(* IEC 61131-3 sources: AXOpen/src/io/app/SystemConstants, 2 files *)

(* ---- plc_line_IoAddresses.st ---- *)
CONFIGURATION IoAddresses
    VAR_GLOBAL

        // Module bnixg35080b5r067/IDM_LinkModule
        bnixg35080b5r067_IDM_LinkModule_BALLUFF_8_Port_IO_Link_Master_Input AT %IB0 : bnixg35080b5r067_IDM_LinkModule_BALLUFF_8_Port_IO_Link_Master_Input_Layout;
        bnixg35080b5r067_IDM_LinkModule_BALLUFF_8_Port_IO_Link_Master_Output AT %QB0 : bnixg35080b5r067_IDM_LinkModule_BALLUFF_8_Port_IO_Link_Master_Output_Layout;
        bnixg35080b5r067_IDM_LinkModule_X01_Input AT %IB1 : bnixg35080b5r067_IDM_LinkModule_X01_Input_Layout;

        // Module et200sp_1/A10
        et200sp_1_A10_Input AT %IB28 : et200sp_1_A10_Input_Layout;

        // Module et200sp_1/A11
        et200sp_1_A11_Input AT %IB26 : et200sp_1_A11_Input_Layout;

        // Module et200sp_1/A12
        et200sp_1_A12_Input AT %IB24 : et200sp_1_A12_Input_Layout;

        // Module et200sp_1/A13
        et200sp_1_A13_Input AT %IB22 : et200sp_1_A13_Input_Layout;

        // Module et200sp_1/A14
        et200sp_1_A14_Input AT %IB20 : et200sp_1_A14_Input_Layout;

        // Module et200sp_1/A15
        et200sp_1_A15_Input AT %IB18 : et200sp_1_A15_Input_Layout;

        // Module et200sp_1/A16
        et200sp_1_A16_Input AT %IB16 : et200sp_1_A16_Input_Layout;

        // Module et200sp_1/A17
        et200sp_1_A17_Input AT %IB14 : et200sp_1_A17_Input_Layout;

        // Module et200sp_1/A20
        et200sp_1_A20_Output AT %QB15 : et200sp_1_A20_Output_Layout;

        // Module et200sp_1/A21
        et200sp_1_A21_Output AT %QB13 : et200sp_1_A21_Output_Layout;

        // Module et200sp_1/A22
        et200sp_1_A22_Output AT %QB11 : et200sp_1_A22_Output_Layout;

        // Module et200sp_1/A23
        et200sp_1_A23_Output AT %QB9 : et200sp_1_A23_Output_Layout;

        // Module et200sp_1/A30
        et200sp_1_A30_Input AT %IB6 : et200sp_1_A30_Input_Layout;

        // Module et200sp_1/A40
        et200sp_1_A40_Output AT %QB1 : et200sp_1_A40_Output_Layout;

        // Module et200sp/A10
        et200sp_A10_Input AT %IB62 : et200sp_A10_Input_Layout;

        // Module et200sp/A20
        et200sp_A20_Output AT %QB49 : et200sp_A20_Output_Layout;

        // Module et200sp/A30
        et200sp_A30_Input AT %IB30 : et200sp_A30_Input_Layout;
        et200sp_A30_Output AT %QB17 : et200sp_A30_Output_Layout;
    END_VAR
END_CONFIGURATION

TYPE
    bnixg35080b5r067_IDM_LinkModule_BALLUFF_8_Port_IO_Link_Master_Input_Layout : STRUCT
        Signals_0 AT %X0.0 : BOOL;
        Signals_1 AT %X0.1 : BOOL;
        Signals_2 AT %X0.2 : BOOL;
        Signals_3 AT %X0.3 : BOOL;
        Signals_4 AT %X0.4 : BOOL;
        Signals_5 AT %X0.5 : BOOL;
        Signals_6 AT %X0.6 : BOOL;
        Signals_7 AT %X0.7 : BOOL;
    END_STRUCT;
END_TYPE

TYPE
    bnixg35080b5r067_IDM_LinkModule_BALLUFF_8_Port_IO_Link_Master_Output_Layout : STRUCT
        Signals_8 AT %X0.0 : BOOL;
        Signals_9 AT %X0.1 : BOOL;
        Signals_10 AT %X0.2 : BOOL;
        Signals_11 AT %X0.3 : BOOL;
        Signals_12 AT %X0.4 : BOOL;
        Signals_13 AT %X0.5 : BOOL;
        Signals_14 AT %X0.6 : BOOL;
        Signals_15 AT %X0.7 : BOOL;
    END_STRUCT;
END_TYPE

TYPE
    bnixg35080b5r067_IDM_LinkModule_X01_Input_Layout : STRUCT
        Signals_0 AT %B0 : ARRAY[0..3] OF BYTE;
        Signals_1 AT %X4.2 : BOOL;
        Signals_2 AT %X4.3 : BOOL;
        Signals_3 AT %X4.4 : BOOL;
        Signals_4 AT %X4.5 : BOOL;
        Signals_5 AT %X4.6 : BOOL;
        Signals_6 AT %X4.7 : BOOL;
    END_STRUCT;
END_TYPE

TYPE
    et200sp_1_A10_Input_Layout : STRUCT
        Signals_0 AT %X0.0 : BOOL;
        Signals_1 AT %X0.1 : BOOL;
        Signals_2 AT %X0.2 : BOOL;
        Signals_3 AT %X0.3 : BOOL;
        Signals_4 AT %X0.4 : BOOL;
        Signals_5 AT %X0.5 : BOOL;
        Signals_6 AT %X0.6 : BOOL;
        Signals_7 AT %X0.7 : BOOL;
        Signals_8 AT %X1.0 : BOOL;
        Signals_9 AT %X1.1 : BOOL;
        Signals_10 AT %X1.2 : BOOL;
        Signals_11 AT %X1.3 : BOOL;
        Signals_12 AT %X1.4 : BOOL;
        Signals_13 AT %X1.5 : BOOL;
        Signals_14 AT %X1.6 : BOOL;
        Signals_15 AT %X1.7 : BOOL;
    END_STRUCT;
END_TYPE

TYPE
    et200sp_1_A11_Input_Layout : STRUCT
        Signals_0 AT %X0.0 : BOOL;
        Signals_1 AT %X0.1 : BOOL;
        Signals_2 AT %X0.2 : BOOL;
        Signals_3 AT %X0.3 : BOOL;
        Signals_4 AT %X0.4 : BOOL;
        Signals_5 AT %X0.5 : BOOL;
        Signals_6 AT %X0.6 : BOOL;
        Signals_7 AT %X0.7 : BOOL;
        Signals_8 AT %X1.0 : BOOL;
        Signals_9 AT %X1.1 : BOOL;
        Signals_10 AT %X1.2 : BOOL;
        Signals_11 AT %X1.3 : BOOL;
        Signals_12 AT %X1.4 : BOOL;
        Signals_13 AT %X1.5 : BOOL;
        Signals_14 AT %X1.6 : BOOL;
        Signals_15 AT %X1.7 : BOOL;
    END_STRUCT;
END_TYPE

TYPE
    et200sp_1_A12_Input_Layout : STRUCT
        Signals_0 AT %X0.0 : BOOL;
        Signals_1 AT %X0.1 : BOOL;
        Signals_2 AT %X0.2 : BOOL;
        Signals_3 AT %X0.3 : BOOL;
        Signals_4 AT %X0.4 : BOOL;
        Signals_5 AT %X0.5 : BOOL;
        Signals_6 AT %X0.6 : BOOL;
        Signals_7 AT %X0.7 : BOOL;
        Signals_8 AT %X1.0 : BOOL;
        Signals_9 AT %X1.1 : BOOL;
        Signals_10 AT %X1.2 : BOOL;
        Signals_11 AT %X1.3 : BOOL;
        Signals_12 AT %X1.4 : BOOL;
        Signals_13 AT %X1.5 : BOOL;
        Signals_14 AT %X1.6 : BOOL;
        Signals_15 AT %X1.7 : BOOL;
    END_STRUCT;
END_TYPE

TYPE
    et200sp_1_A13_Input_Layout : STRUCT
        Signals_0 AT %X0.0 : BOOL;
        Signals_1 AT %X0.1 : BOOL;
        Signals_2 AT %X0.2 : BOOL;
        Signals_3 AT %X0.3 : BOOL;
        Signals_4 AT %X0.4 : BOOL;
        Signals_5 AT %X0.5 : BOOL;
        Signals_6 AT %X0.6 : BOOL;
        Signals_7 AT %X0.7 : BOOL;
        Signals_8 AT %X1.0 : BOOL;
        Signals_9 AT %X1.1 : BOOL;
        Signals_10 AT %X1.2 : BOOL;
        Signals_11 AT %X1.3 : BOOL;
        Signals_12 AT %X1.4 : BOOL;
        Signals_13 AT %X1.5 : BOOL;
        Signals_14 AT %X1.6 : BOOL;
        Signals_15 AT %X1.7 : BOOL;
    END_STRUCT;
END_TYPE

TYPE
    et200sp_1_A14_Input_Layout : STRUCT
        Signals_0 AT %X0.0 : BOOL;
        Signals_1 AT %X0.1 : BOOL;
        Signals_2 AT %X0.2 : BOOL;
        Signals_3 AT %X0.3 : BOOL;
        Signals_4 AT %X0.4 : BOOL;
        Signals_5 AT %X0.5 : BOOL;
        Signals_6 AT %X0.6 : BOOL;
        Signals_7 AT %X0.7 : BOOL;
        Signals_8 AT %X1.0 : BOOL;
        Signals_9 AT %X1.1 : BOOL;
        Signals_10 AT %X1.2 : BOOL;
        Signals_11 AT %X1.3 : BOOL;
        Signals_12 AT %X1.4 : BOOL;
        Signals_13 AT %X1.5 : BOOL;
        Signals_14 AT %X1.6 : BOOL;
        Signals_15 AT %X1.7 : BOOL;
    END_STRUCT;
END_TYPE

TYPE
    et200sp_1_A15_Input_Layout : STRUCT
        Signals_0 AT %X0.0 : BOOL;
        Signals_1 AT %X0.1 : BOOL;
        Signals_2 AT %X0.2 : BOOL;
        Signals_3 AT %X0.3 : BOOL;
        Signals_4 AT %X0.4 : BOOL;
        Signals_5 AT %X0.5 : BOOL;
        Signals_6 AT %X0.6 : BOOL;
        Signals_7 AT %X0.7 : BOOL;
        Signals_8 AT %X1.0 : BOOL;
        Signals_9 AT %X1.1 : BOOL;
        Signals_10 AT %X1.2 : BOOL;
        Signals_11 AT %X1.3 : BOOL;
        Signals_12 AT %X1.4 : BOOL;
        Signals_13 AT %X1.5 : BOOL;
        Signals_14 AT %X1.6 : BOOL;
        Signals_15 AT %X1.7 : BOOL;
    END_STRUCT;
END_TYPE

TYPE
    et200sp_1_A16_Input_Layout : STRUCT
        Signals_0 AT %X0.0 : BOOL;
        Signals_1 AT %X0.1 : BOOL;
        Signals_2 AT %X0.2 : BOOL;
        Signals_3 AT %X0.3 : BOOL;
        Signals_4 AT %X0.4 : BOOL;
        Signals_5 AT %X0.5 : BOOL;
        Signals_6 AT %X0.6 : BOOL;
        Signals_7 AT %X0.7 : BOOL;
        Signals_8 AT %X1.0 : BOOL;
        Signals_9 AT %X1.1 : BOOL;
        Signals_10 AT %X1.2 : BOOL;
        Signals_11 AT %X1.3 : BOOL;
        Signals_12 AT %X1.4 : BOOL;
        Signals_13 AT %X1.5 : BOOL;
        Signals_14 AT %X1.6 : BOOL;
        Signals_15 AT %X1.7 : BOOL;
    END_STRUCT;
END_TYPE

TYPE
    et200sp_1_A17_Input_Layout : STRUCT
        Signals_0 AT %X0.0 : BOOL;
        Signals_1 AT %X0.1 : BOOL;
        Signals_2 AT %X0.2 : BOOL;
        Signals_3 AT %X0.3 : BOOL;
        Signals_4 AT %X0.4 : BOOL;
        Signals_5 AT %X0.5 : BOOL;
        Signals_6 AT %X0.6 : BOOL;
        Signals_7 AT %X0.7 : BOOL;
        Signals_8 AT %X1.0 : BOOL;
        Signals_9 AT %X1.1 : BOOL;
        Signals_10 AT %X1.2 : BOOL;
        Signals_11 AT %X1.3 : BOOL;
        Signals_12 AT %X1.4 : BOOL;
        Signals_13 AT %X1.5 : BOOL;
        Signals_14 AT %X1.6 : BOOL;
        Signals_15 AT %X1.7 : BOOL;
    END_STRUCT;
END_TYPE

TYPE
    et200sp_1_A20_Output_Layout : STRUCT
        Signals_0 AT %X0.0 : BOOL;
        Signals_1 AT %X0.1 : BOOL;
        Signals_2 AT %X0.2 : BOOL;
        Signals_3 AT %X0.3 : BOOL;
        Signals_4 AT %X0.4 : BOOL;
        Signals_5 AT %X0.5 : BOOL;
        Signals_6 AT %X0.6 : BOOL;
        Signals_7 AT %X0.7 : BOOL;
        Signals_8 AT %X1.0 : BOOL;
        Signals_9 AT %X1.1 : BOOL;
        Signals_10 AT %X1.2 : BOOL;
        Signals_11 AT %X1.3 : BOOL;
        Signals_12 AT %X1.4 : BOOL;
        Signals_13 AT %X1.5 : BOOL;
        Signals_14 AT %X1.6 : BOOL;
        Signals_15 AT %X1.7 : BOOL;
    END_STRUCT;
END_TYPE

TYPE
    et200sp_1_A21_Output_Layout : STRUCT
        Signals_0 AT %X0.0 : BOOL;
        Signals_1 AT %X0.1 : BOOL;
        Signals_2 AT %X0.2 : BOOL;
        Signals_3 AT %X0.3 : BOOL;
        Signals_4 AT %X0.4 : BOOL;
        Signals_5 AT %X0.5 : BOOL;
        Signals_6 AT %X0.6 : BOOL;
        Signals_7 AT %X0.7 : BOOL;
        Signals_8 AT %X1.0 : BOOL;
        Signals_9 AT %X1.1 : BOOL;
        Signals_10 AT %X1.2 : BOOL;
        Signals_11 AT %X1.3 : BOOL;
        Signals_12 AT %X1.4 : BOOL;
        Signals_13 AT %X1.5 : BOOL;
        Signals_14 AT %X1.6 : BOOL;
        Signals_15 AT %X1.7 : BOOL;
    END_STRUCT;
END_TYPE

TYPE
    et200sp_1_A22_Output_Layout : STRUCT
        Signals_0 AT %X0.0 : BOOL;
        Signals_1 AT %X0.1 : BOOL;
        Signals_2 AT %X0.2 : BOOL;
        Signals_3 AT %X0.3 : BOOL;
        Signals_4 AT %X0.4 : BOOL;
        Signals_5 AT %X0.5 : BOOL;
        Signals_6 AT %X0.6 : BOOL;
        Signals_7 AT %X0.7 : BOOL;
        Signals_8 AT %X1.0 : BOOL;
        Signals_9 AT %X1.1 : BOOL;
        Signals_10 AT %X1.2 : BOOL;
        Signals_11 AT %X1.3 : BOOL;
        Signals_12 AT %X1.4 : BOOL;
        Signals_13 AT %X1.5 : BOOL;
        Signals_14 AT %X1.6 : BOOL;
        Signals_15 AT %X1.7 : BOOL;
    END_STRUCT;
END_TYPE

TYPE
    et200sp_1_A23_Output_Layout : STRUCT
        Signals_0 AT %X0.0 : BOOL;
        Signals_1 AT %X0.1 : BOOL;
        Signals_2 AT %X0.2 : BOOL;
        Signals_3 AT %X0.3 : BOOL;
        Signals_4 AT %X0.4 : BOOL;
        Signals_5 AT %X0.5 : BOOL;
        Signals_6 AT %X0.6 : BOOL;
        Signals_7 AT %X0.7 : BOOL;
        Signals_8 AT %X1.0 : BOOL;
        Signals_9 AT %X1.1 : BOOL;
        Signals_10 AT %X1.2 : BOOL;
        Signals_11 AT %X1.3 : BOOL;
        Signals_12 AT %X1.4 : BOOL;
        Signals_13 AT %X1.5 : BOOL;
        Signals_14 AT %X1.6 : BOOL;
        Signals_15 AT %X1.7 : BOOL;
    END_STRUCT;
END_TYPE

TYPE
    et200sp_1_A30_Input_Layout : STRUCT
        Signals_0 AT %B0 : INT;
        Signals_1 AT %B2 : INT;
        Signals_2 AT %B4 : INT;
        Signals_3 AT %B6 : INT;
    END_STRUCT;
END_TYPE

TYPE
    et200sp_1_A40_Output_Layout : STRUCT
        Signals_0 AT %B0 : INT;
        Signals_1 AT %B2 : INT;
        Signals_2 AT %B4 : INT;
        Signals_3 AT %B6 : INT;
    END_STRUCT;
END_TYPE

TYPE
    et200sp_A10_Input_Layout : STRUCT
        Signals_0 AT %X0.0 : BOOL;
        Signals_1 AT %X0.1 : BOOL;
        Signals_2 AT %X0.2 : BOOL;
        Signals_3 AT %X0.3 : BOOL;
        Signals_4 AT %X0.4 : BOOL;
        Signals_5 AT %X0.5 : BOOL;
        Signals_6 AT %X0.6 : BOOL;
        Signals_7 AT %X0.7 : BOOL;
        Signals_8 AT %X1.0 : BOOL;
        Signals_9 AT %X1.1 : BOOL;
        Signals_10 AT %X1.2 : BOOL;
        Signals_11 AT %X1.3 : BOOL;
        Signals_12 AT %X1.4 : BOOL;
        Signals_13 AT %X1.5 : BOOL;
        Signals_14 AT %X1.6 : BOOL;
        Signals_15 AT %X1.7 : BOOL;
    END_STRUCT;
END_TYPE

TYPE
    et200sp_A20_Output_Layout : STRUCT
        Signals_0 AT %X0.0 : BOOL;
        Signals_1 AT %X0.1 : BOOL;
        Signals_2 AT %X0.2 : BOOL;
        Signals_3 AT %X0.3 : BOOL;
        Signals_4 AT %X0.4 : BOOL;
        Signals_5 AT %X0.5 : BOOL;
        Signals_6 AT %X0.6 : BOOL;
        Signals_7 AT %X0.7 : BOOL;
        Signals_8 AT %X1.0 : BOOL;
        Signals_9 AT %X1.1 : BOOL;
        Signals_10 AT %X1.2 : BOOL;
        Signals_11 AT %X1.3 : BOOL;
        Signals_12 AT %X1.4 : BOOL;
        Signals_13 AT %X1.5 : BOOL;
        Signals_14 AT %X1.6 : BOOL;
        Signals_15 AT %X1.7 : BOOL;
    END_STRUCT;
END_TYPE

TYPE
    et200sp_A30_Input_Layout : STRUCT
        Signals_0 AT %B0 : BYTE;
        Signals_1 AT %B1 : BYTE;
        Signals_2 AT %B2 : BYTE;
        Signals_3 AT %B3 : BYTE;
        Signals_4 AT %B4 : BYTE;
        Signals_5 AT %B5 : BYTE;
        Signals_6 AT %B6 : BYTE;
        Signals_7 AT %B7 : BYTE;
        Signals_8 AT %B8 : BYTE;
        Signals_9 AT %B9 : BYTE;
        Signals_10 AT %B10 : BYTE;
        Signals_11 AT %B11 : BYTE;
        Signals_12 AT %B12 : BYTE;
        Signals_13 AT %B13 : BYTE;
        Signals_14 AT %B14 : BYTE;
        Signals_15 AT %B15 : BYTE;
        Signals_16 AT %B16 : BYTE;
        Signals_17 AT %B17 : BYTE;
        Signals_18 AT %B18 : BYTE;
        Signals_19 AT %B19 : BYTE;
        Signals_20 AT %B20 : BYTE;
        Signals_21 AT %B21 : BYTE;
        Signals_22 AT %B22 : BYTE;
        Signals_23 AT %B23 : BYTE;
        Signals_24 AT %B24 : BYTE;
        Signals_25 AT %B25 : BYTE;
        Signals_26 AT %B26 : BYTE;
        Signals_27 AT %B27 : BYTE;
        Signals_28 AT %B28 : BYTE;
        Signals_29 AT %B29 : BYTE;
        Signals_30 AT %B30 : BYTE;
        Signals_31 AT %B31 : BYTE;
    END_STRUCT;
END_TYPE

TYPE
    et200sp_A30_Output_Layout : STRUCT
        Signals_32 AT %B0 : BYTE;
        Signals_33 AT %B1 : BYTE;
        Signals_34 AT %B2 : BYTE;
        Signals_35 AT %B3 : BYTE;
        Signals_36 AT %B4 : BYTE;
        Signals_37 AT %B5 : BYTE;
        Signals_38 AT %B6 : BYTE;
        Signals_39 AT %B7 : BYTE;
        Signals_40 AT %B8 : BYTE;
        Signals_41 AT %B9 : BYTE;
        Signals_42 AT %B10 : BYTE;
        Signals_43 AT %B11 : BYTE;
        Signals_44 AT %B12 : BYTE;
        Signals_45 AT %B13 : BYTE;
        Signals_46 AT %B14 : BYTE;
        Signals_47 AT %B15 : BYTE;
        Signals_48 AT %B16 : BYTE;
        Signals_49 AT %B17 : BYTE;
        Signals_50 AT %B18 : BYTE;
        Signals_51 AT %B19 : BYTE;
        Signals_52 AT %B20 : BYTE;
        Signals_53 AT %B21 : BYTE;
        Signals_54 AT %B22 : BYTE;
        Signals_55 AT %B23 : BYTE;
        Signals_56 AT %B24 : BYTE;
        Signals_57 AT %B25 : BYTE;
        Signals_58 AT %B26 : BYTE;
        Signals_59 AT %B27 : BYTE;
        Signals_60 AT %B28 : BYTE;
        Signals_61 AT %B29 : BYTE;
        Signals_62 AT %B30 : BYTE;
        Signals_63 AT %B31 : BYTE;
    END_STRUCT;
END_TYPE

(* ---- plc_line_HwIdentifiers.st ---- *)
CONFIGURATION HardwareIDs
    VAR_GLOBAL CONSTANT
        bni00l3_2_HwID : UINT := UINT#258;
        bni00l3_2_16_DI_HwID : UINT := UINT#263;
        bni00l3_2_16_DI_BALLUFF_8_Port_IO_Link_Master_HwID : UINT := UINT#264;
        bni00l3_2_Rack_HwID : UINT := UINT#261;
        bni00l3_2_X01_HwID : UINT := UINT#265;
        bni00l3_2_X02_HwID : UINT := UINT#266;
        bni00l3_2_X03_HwID : UINT := UINT#267;
        bni00l3_2_X04_HwID : UINT := UINT#268;
        bni00l3_2_X05_HwID : UINT := UINT#269;
        bni00l3_2_X06_HwID : UINT := UINT#270;
        bni00l3_2_X07_HwID : UINT := UINT#271;
        bni00l3_2_X08_HwID : UINT := UINT#272;
        bni00l3_2_bni00l3_2_HwID : UINT := UINT#262;
        bni00l3_2_bni00l3_2_BNI_XG3_508_0B5_R067_HwID : UINT := UINT#273;
        bni00l3_2_bni00l3_2_PN_IO_HwID : UINT := UINT#257;
        bni00l3_2_bni00l3_2_PN_IO_Port_1_HwID : UINT := UINT#259;
        bni00l3_2_bni00l3_2_PN_IO_Port_2_HwID : UINT := UINT#260;
        et200sp_HwID : UINT := UINT#276;
        et200sp_A100_Server_module_V1_1_0_bytes_HwID : UINT := UINT#281;
        et200sp_A10_DI_16x24VDC_ST_V1_1_HwID : UINT := UINT#284;
        et200sp_A20_DQ_16x24VDC_0_5A_ST_V1_1_HwID : UINT := UINT#283;
        et200sp_A30_CM_4xIO_Link_V2_2_32I_32O_HwID : UINT := UINT#282;
        et200sp_Rack_HwID : UINT := UINT#279;
        et200sp_et200sp_HwID : UINT := UINT#280;
        et200sp_et200sp_IM_155_6_PN_ST_V4_2_HwID : UINT := UINT#285;
        et200sp_et200sp_PN_IO_HwID : UINT := UINT#275;
        et200sp_et200sp_Port_1_HwID : UINT := UINT#277;
        et200sp_et200sp_Port_2_HwID : UINT := UINT#278;
        plc_line_HwID : UINT := UINT#32;
        plc_line_Rail_0_HwID : UINT := UINT#286;
        plc_line_plc_line_HwID : UINT := UINT#48;
        plc_line_plc_line_CPU_display_1_HwID : UINT := UINT#54;
        plc_line_plc_line_Card_reader_writer_1_HwID : UINT := UINT#51;
        plc_line_plc_line_DP_interface_1_HwID : UINT := UINT#60;
        plc_line_plc_line_OPC_UA_1_HwID : UINT := UINT#117;
        plc_line_plc_line_PROFINET_interface_1_HwID : UINT := UINT#64;
        plc_line_plc_line_PROFINET_interface_1_Port_1_HwID : UINT := UINT#65;
        plc_line_plc_line_PROFINET_interface_1_Port_2_HwID : UINT := UINT#66;
        plc_line_plc_line_PROFINET_interface_2_HwID : UINT := UINT#72;
        plc_line_plc_line_PROFINET_interface_2_Port_3_HwID : UINT := UINT#73;
        plc_line_plc_line_Virtual_communication_interface_HwID : UINT := UINT#135;
        profinet2_plc_line_HwID : UINT := UINT#256;
        profinet_plc_line_HwID : UINT := UINT#274;

    END_VAR
END_CONFIGURATION
